Staubli VAL3: getDistance.pgx

public program getDistance(tool x_tTool, num& x_nDistance[], bool x_bCycle, num x_nIndex)
  local num l_nDistance
  local point l_pPoint
  local num l_nValue
  local trsf l_trsfEmpty
begin
  // first point
  if x_nIndex==0
    x_nDistance=10
    return
  elseIf x_bCycle
    // an other one
    x_nDistance=distance(jointToPoint(x_tTool,world,pt:tTraj[sTrajCycle].tData[x_nIndex-1].jJoint),jointToPoint(x_tTool,world,pt:tTraj[sTrajCycle].tData[x_nIndex].jJoint))
  else
     x_nDistance=distance(jointToPoint(x_tTool,world,jEditPoint.tData[x_nIndex-1].jJoint),jointToPoint(x_tTool,world,jEditPoint.tData[x_nIndex].jJoint))
  endIf
end
